Universal Robots URScript: 2024DragonThickMarker.script

def unnamed():
  set_target_payload(1.070000, [0.002000, 0.003000, 0.057000], [0.001723, 0.001723, 0.001723, 0.000000, 0.000000, 0.000000])
  set_tool_communication(True, 1000000, 2, 1, 1.5, 3.5)
  set_tool_output_mode(0)
  set_tool_digital_output_mode(0, 1)
  set_tool_digital_output_mode(1, 1)
  set_tool_voltage(0)
  set_standard_analog_input_domain(0, 1)
  set_standard_analog_input_domain(1, 1)
  set_tool_analog_input_domain(0, 1)
  set_tool_analog_input_domain(1, 1)
  set_analog_outputdomain(0, 0)
  set_analog_outputdomain(1, 0)
  set_input_actions_to_default()
  step_count_120ef5ed_3093_42e9_8e41_c6a461b1e92a = 0.0
  thread Step_Counter_Thread_6ab2a575_f1a7_416e_8c30_f36541ff69b0():
    while (True):
      step_count_120ef5ed_3093_42e9_8e41_c6a461b1e92a = step_count_120ef5ed_3093_42e9_8e41_c6a461b1e92a + 1.0
      sync()
    end
  end
  run Step_Counter_Thread_6ab2a575_f1a7_416e_8c30_f36541ff69b0()
  set_tcp(p[0.0,0.0,0.0,0.0,0.0,0.0])
  set_gravity([0.0, 0.0, 9.82])
  set_safety_mode_transition_hardness(1)
  global Plane_1=p[-0.700006141123905,1.3454883874109249E-6,0.3910559577028425,-1.2089868272251132,-1.2089999932245832,1.20858562628424]
  global Plane_2=p[0.0,0.0,0.0,0.0,0.0,0.0]
  global Point_1=p[0.6913645118948067,-0.12399382748223003,0.49223711947071,-1.2983729986843258,1.1259514972191385,-1.2203503861141718]
  $ 1 "Robot Program"
  $ 2 "Script: 2024Dagonv3_1_marker.script"
  def Machining1():
    # Default parameters:
    global speed_ms = 0.3
    global speed_rads = 0.75
    global accel_mss = 3
    global accel_radss = 1.2
    global blend_radius_m = 0.001

    # Add subprograms here
    # Start of main program
    # Program generated by RoboDK v5.6.5 for UR10e on 12/01/2024 12:52:10
    # Using nominal kinematics.
    blend_radius_m = 0.000
    speed_ms = 1.000
    # set_reference(p[0.335000, -0.152000, -0.035000, 0.000000, 0.000000, 0.000000])
    set_tcp(p[0.000000, 0.000000, 0.252000, 0.000000, 0.000000, 0.000000])
    # Show Tool
    movej([0.067194, -1.029625, -2.540120, -1.142644, 1.570796, 1.637990],accel_radss,speed_rads,0,blend_radius_m)
    movel([0.067194, -1.029625, -2.540120, -1.142644, 1.570796, 1.637990],accel_mss,speed_ms,0,blend_radius_m)
    # Splitting Linear movement in 22 (instruction 7: MoveL 3)
    movel([0.067194, -1.035168, -2.546706, -1.130514, 1.570796, 1.637990],accel_mss,speed_ms,0,blend_radius_m)
    movel([0.067194, -1.040913, -2.553250, -1.118226, 1.570796, 1.637990],accel_mss,speed_ms,0,blend_radius_m)
    movel([0.067194, -1.046863, -2.559752, -1.105774, 1.570796, 1.637990],accel_mss,speed_ms,0,blend_radius_m)
    movel([0.067194, -1.053024, -2.566210, -1.093155, 1.570796, 1.637990],accel_mss,speed_ms,0,blend_radius_m)
    movel([0.067194, -1.059401, -2.572624, -1.080365, 1.570796, 1.637990],accel_mss,speed_ms,0,blend_radius_m)
    movel([0.067194, -1.065999, -2.578992, -1.067399, 1.570796, 1.637990],accel_mss,speed_ms,0,blend_radius_m)
    movel([0.067194, -1.072824, -2.585312, -1.054253, 1.570796, 1.637990],accel_mss,speed_ms,0,blend_radius_m)
    movel([0.067194, -1.079881, -2.591585, -1.040923, 1.570796, 1.637990],accel_mss,speed_ms,0,blend_radius_m)
    movel([0.067194, -1.087175, -2.597809, -1.027405, 1.570796, 1.637990],accel_mss,speed_ms,0,blend_radius_m)
    movel([0.067194, -1.094713, -2.603982, -1.013694, 1.570796, 1.637990],accel_mss,speed_ms,0,blend_radius_m)
    movel([0.067194, -1.102499, -2.610103, -0.999786, 1.570796, 1.637990],accel_mss,speed_ms,0,blend_radius_m)
    movel([0.067194, -1.110540, -2.616171, -0.985677, 1.570796, 1.637990],accel_mss,speed_ms,0,blend_radius_m)
    movel([0.067194, -1.118842, -2.622185, -0.971363, 1.570796, 1.637990],accel_mss,speed_ms,0,blend_radius_m)
    movel([0.067194, -1.127410, -2.628141, -0.956838, 1.570796, 1.637990],accel_mss,speed_ms,0,blend_radius_m)
    movel([0.067194, -1.136249, -2.634040, -0.942099, 1.570796, 1.637990],accel_mss,speed_ms,0,blend_radius_m)
    movel([0.067194, -1.145367, -2.639880, -0.927142, 1.570796, 1.637990],accel_mss,speed_ms,0,blend_radius_m)
    movel([0.067194, -1.154769, -2.645658, -0.911961, 1.570796, 1.637990],accel_mss,speed_ms,0,blend_radius_m)
    movel([0.067194, -1.164461, -2.651374, -0.896554, 1.570796, 1.637990],accel_mss,speed_ms,0,blend_radius_m)
    movel([0.067194, -1.174449, -2.657024, -0.880916, 1.570796, 1.637990],accel_mss,speed_ms,0,blend_radius_m)
    movel([0.067194, -1.184738, -2.662608, -0.865043, 1.570796, 1.637990],accel_mss,speed_ms,0,blend_radius_m)
    movel([0.067194, -1.195335, -2.668122, -0.848931, 1.570796, 1.637990],accel_mss,speed_ms,0,blend_radius_m)
    movel([0.067194, -1.206246, -2.673566, -0.832577, 1.570796, 1.637990],accel_mss,speed_ms,0,blend_radius_m)
    movel([0.067194, -1.206246, -2.673566, -0.832577, 1.570796, 1.637990],accel_mss,speed_ms,0,blend_radius_m)
    speed_ms = 1.000
    movel([0.067194, -1.206246, -2.673566, -0.832577, 1.570796, 1.637990],accel_mss,speed_ms,0,blend_radius_m)
    movel([0.067194, -1.206246, -2.673566, -0.832577, 1.570796, 1.637990],accel_mss,speed_ms,0,blend_radius_m)
    movel([0.067194, -1.206246, -2.673566, -0.832577, 1.570796, 1.637990],accel_mss,speed_ms,0,blend_radius_m)
    speed_ms = 0.005
    # Splitting Linear movement in 4 (instruction 14: MoveL 8)
    movel([0.067194, -1.194262, -2.667574, -0.850553, 1.570796, 1.637990],accel_mss,speed_ms,0,blend_radius_m)
    movel([0.067194, -1.182656, -2.661496, -0.868237, 1.570796, 1.637990],accel_mss,speed_ms,0,blend_radius_m)
    movel([0.067194, -1.171421, -2.655336, -0.885632, 1.570796, 1.637990],accel_mss,speed_ms,0,blend_radius_m)
    movel([0.067194, -1.160549, -2.649095, -0.902745, 1.570796, 1.637990],accel_mss,speed_ms,0,blend_radius_m)
    speed_ms = 1.000
    # Splitting Linear movement in 4 (instruction 16: MoveL 9)
    movel([0.067194, -1.171421, -2.655336, -0.885632, 1.570796, 1.637990],accel_mss,speed_ms,0,blend_radius_m)
    movel([0.067194, -1.182656, -2.661496, -0.868237, 1.570796, 1.637990],accel_mss,speed_ms,0,blend_radius_m)
    movel([0.067194, -1.194262, -2.667574, -0.850553, 1.570796, 1.637990],accel_mss,speed_ms,0,blend_radius_m)
    movel([0.067194, -1.206246, -2.673566, -0.832577, 1.570796, 1.637990],accel_mss,speed_ms,0,blend_radius_m)
    speed_ms = 0.040
    movel([0.067194, -1.206246, -2.673566, -0.832577, 1.570796, 1.637990],accel_mss,speed_ms,0,blend_radius_m)
    speed_ms = 1.000
    movel([0.067194, -1.206246, -2.673566, -0.832577, 1.570796, 1.637990],accel_mss,speed_ms,0,blend_radius_m)
    # Splitting Linear movement in 12 (instruction 21: MoveL 12)
    movel([0.077689, -1.208311, -2.672566, -0.831512, 1.570796, 1.648485],accel_mss,speed_ms,0,blend_radius_m)
    movel([0.088074, -1.210516, -2.671493, -0.830380, 1.570796, 1.658871],accel_mss,speed_ms,0,blend_radius_m)
    movel([0.098348, -1.212858, -2.670347, -0.829184, 1.570796, 1.669145],accel_mss,speed_ms,0,blend_radius_m)
    movel([0.108510, -1.215333, -2.669129, -0.827926, 1.570796, 1.679306],accel_mss,speed_ms,0,blend_radius_m)
    movel([0.118557, -1.217940, -2.667840, -0.826610, 1.570796, 1.689354],accel_mss,speed_ms,0,blend_radius_m)
    movel([0.128491, -1.220675, -2.666478, -0.825236, 1.570796, 1.699287],accel_mss,speed_ms,0,blend_radius_m)
    movel([0.138308, -1.223537, -2.665044, -0.823808, 1.570796, 1.709104],accel_mss,speed_ms,0,blend_radius_m)
    movel([0.148009, -1.226521, -2.663539, -0.822329, 1.570796, 1.718806],accel_mss,speed_ms,0,blend_radius_m)
    movel([0.157594, -1.229625, -2.661962, -0.820802, 1.570796, 1.728390],accel_mss,speed_ms,0,blend_radius_m)
    movel([0.167061, -1.232845, -2.660315, -0.819229, 1.570796, 1.737857],accel_mss,speed_ms,0,blend_radius_m)
    movel([0.176410, -1.236179, -2.658597, -0.817613, 1.570796, 1.747207],accel_mss,speed_ms,0,blend_radius_m)
    movel([0.185641, -1.239624, -2.656808, -0.815957, 1.570796, 1.756438],accel_mss,speed_ms,0,blend_radius_m)
    speed_ms = 0.005
    # Splitting Linear movement in 4 (instruction 23: MoveL 13)
    movel([0.185641, -1.251804, -2.662521, -0.798064, 1.570796, 1.756438],accel_mss,speed_ms,0,blend_radius_m)
    movel([0.185641, -1.264347, -2.668140, -0.779901, 1.570796, 1.756438],accel_mss,speed_ms,0,blend_radius_m)
    movel([0.185641, -1.277260, -2.673664, -0.761465, 1.570796, 1.756438],accel_mss,speed_ms,0,blend_radius_m)
    movel([0.185641, -1.290546, -2.679089, -0.742755, 1.570796, 1.756438],accel_mss,speed_ms,0,blend_radius_m)
    speed_ms = 0.035
    movel([0.190535, -1.290094, -2.679342, -0.742953, 1.570796, 1.761331],accel_mss,speed_ms,0,blend_radius_m)
    movel([0.192211, -1.292754, -2.677845, -0.741789, 1.570796, 1.763007],accel_mss,speed_ms,0,blend_radius_m)
    movel([0.190799, -1.296821, -2.675539, -0.740029, 1.570796, 1.761596],accel_mss,speed_ms,0,blend_radius_m)
    movel([0.186440, -1.300624, -2.673363, -0.738402, 1.570796, 1.757236],accel_mss,speed_ms,0,blend_radius_m)
    speed_ms = 0.005
    movel([0.186440, -1.290042, -2.669080, -0.753268, 1.570796, 1.757236],accel_mss,speed_ms,0,blend_radius_m)
    speed_ms = 0.040
    # Splitting Linear movement in 2 (instruction 32: MoveL 19)
    movel([0.192451, -1.282070, -2.673547, -0.756771, 1.570796, 1.763248],accel_mss,speed_ms,0,blend_radius_m)
    movel([0.198560, -1.273987, -2.677995, -0.760408, 1.570796, 1.769357],accel_mss,speed_ms,0,blend_radius_m)
    speed_ms = 0.005
    movel([0.198560, -1.284689, -2.682355, -0.745345, 1.570796, 1.769357],accel_mss,speed_ms,0,blend_radius_m)
    speed_ms = 0.035
    movel([0.198826, -1.280371, -2.684734, -0.747284, 1.570796, 1.769623],accel_mss,speed_ms,0,blend_radius_m)
    movel([0.195615, -1.278404, -2.685810, -0.748175, 1.570796, 1.766412],accel_mss,speed_ms,0,blend_radius_m)
    movel([0.188967, -1.279617, -2.685147, -0.747625, 1.570796, 1.759764],accel_mss,speed_ms,0,blend_radius_m)
    movel([0.185695, -1.277747, -2.686168, -0.748474, 1.570796, 1.756491],accel_mss,speed_ms,0,blend_radius_m)
    movel([0.186358, -1.274154, -2.688117, -0.750117, 1.570796, 1.757155],accel_mss,speed_ms,0,blend_radius_m)
    movel([0.189422, -1.271170, -2.689724, -0.751495, 1.570796, 1.760218],accel_mss,speed_ms,0,blend_radius_m)
    movel([0.193300, -1.271190, -2.689713, -0.751486, 1.570796, 1.764097],accel_mss,speed_ms,0,blend_radius_m)
    speed_ms = 0.005
    movel([0.193300, -1.260391, -2.685288, -0.766710, 1.570796, 1.764097],accel_mss,speed_ms,0,blend_radius_m)
    speed_ms = 0.040
    # Splitting Linear movement in 4 (instruction 46: MoveL 29)
    movel([0.178839, -1.264011, -2.683369, -0.765009, 1.570796, 1.749636],accel_mss,speed_ms,0,blend_radius_m)
    movel([0.164394, -1.267779, -2.681354, -0.763257, 1.570796, 1.735191],accel_mss,speed_ms,0,blend_radius_m)
    movel([0.149972, -1.271689, -2.679243, -0.761456, 1.570796, 1.720768],accel_mss,speed_ms,0,blend_radius_m)
    movel([0.135577, -1.275738, -2.677038, -0.759613, 1.570796, 1.706373],accel_mss,speed_ms,0,blend_radius_m)
    speed_ms = 0.005
    movel([0.135577, -1.286427, -2.681390, -0.744572, 1.570796, 1.706373],accel_mss,speed_ms,0,blend_radius_m)
    speed_ms = 0.035
    # Splitting Linear movement in 4 (instruction 50: MoveL 31)
    movel([0.144537, -1.281430, -2.684152, -0.746806, 1.570796, 1.715333],accel_mss,speed_ms,0,blend_radius_m)
    movel([0.153562, -1.276433, -2.686883, -0.749073, 1.570796, 1.724358],accel_mss,speed_ms,0,blend_radius_m)
    movel([0.162651, -1.271435, -2.689582, -0.751372, 1.570796, 1.733448],accel_mss,speed_ms,0,blend_radius_m)
    movel([0.171806, -1.266439, -2.692248, -0.753702, 1.570796, 1.742602],accel_mss,speed_ms,0,blend_radius_m)
    # Splitting Linear movement in 2 (instruction 51: MoveL 32)
    movel([0.180931, -1.259543, -2.695876, -0.756970, 1.570796, 1.751728],accel_mss,speed_ms,0,blend_radius_m)
    movel([0.190162, -1.252594, -2.699472, -0.760323, 1.570796, 1.760958],accel_mss,speed_ms,0,blend_radius_m)
    speed_ms = 0.005
    movel([0.190162, -1.241669, -2.694957, -0.775763, 1.570796, 1.760958],accel_mss,speed_ms,0,blend_radius_m)
    speed_ms = 0.040
    # Splitting Linear movement in 8 (instruction 55: MoveL 34)
    movel([0.177847, -1.248567, -2.691444, -0.772378, 1.570796, 1.748643],accel_mss,speed_ms,0,blend_radius_m)
    movel([0.165650, -1.255464, -2.687874, -0.769051, 1.570796, 1.736446],accel_mss,speed_ms,0,blend_radius_m)
    movel([0.153572, -1.262358, -2.684247, -0.765784, 1.570796, 1.724369],accel_mss,speed_ms,0,blend_radius_m)
    movel([0.141614, -1.269247, -2.680564, -0.762579, 1.570796, 1.712411],accel_mss,speed_ms,0,blend_radius_m)
    movel([0.129776, -1.276127, -2.676825, -0.759437, 1.570796, 1.700573],accel_mss,speed_ms,0,blend_radius_m)
    movel([0.118059, -1.282997, -2.673032, -0.756360, 1.570796, 1.688856],accel_mss,speed_ms,0,blend_radius_m)
    movel([0.106463, -1.289855, -2.669185, -0.753349, 1.570796, 1.677259],accel_mss,speed_ms,0,blend_radius_m)
    movel([0.094987, -1.296699, -2.665285, -0.750405, 1.570796, 1.665784],accel_mss,speed_ms,0,blend_radius_m)
    speed_ms = 0.005
    movel([0.094987, -1.307230, -2.669536, -0.735623, 1.570796, 1.665784],accel_mss,speed_ms,0,blend_radius_m)
    speed_ms = 0.035
    movel([0.101831, -1.302246, -2.672429, -0.737715, 1.570796, 1.672627],accel_mss,speed_ms,0,blend_radius_m)
    movel([0.103479, -1.304486, -2.671133, -0.736771, 1.570796, 1.674276],accel_mss,speed_ms,0,blend_radius_m)
    movel([0.102130, -1.311236, -2.667187, -0.733966, 1.570796, 1.672926],accel_mss,speed_ms,0,blend_radius_m)
    # Splitting Linear movement in 2 (instruction 62: MoveL 39)
    movel([0.109636, -1.305912, -2.670304, -0.736173, 1.570796, 1.680433],accel_mss,speed_ms,0,blend_radius_m)
    movel([0.117212, -1.300561, -2.673399, -0.738429, 1.570796, 1.688008],accel_mss,speed_ms,0,blend_radius_m)
    movel([0.121435, -1.299795, -2.673839, -0.738755, 1.570796, 1.692231],accel_mss,speed_ms,0,blend_radius_m)
    speed_ms = 0.005
    movel([0.121435, -1.289206, -2.669552, -0.753631, 1.570796, 1.692231],accel_mss,speed_ms,0,blend_radius_m)
    speed_ms = 0.040
    movel([0.111114, -1.287406, -2.670566, -0.754417, 1.570796, 1.681910],accel_mss,speed_ms,0,blend_radius_m)
    speed_ms = 0.005
    movel([0.111114, -1.298008, -2.674862, -0.739519, 1.570796, 1.681910],accel_mss,speed_ms,0,blend_radius_m)
    speed_ms = 0.035
    movel([0.111474, -1.294449, -2.676887, -0.741053, 1.570796, 1.682270],accel_mss,speed_ms,0,blend_radius_m)
    movel([0.115727, -1.290498, -2.679115, -0.742775, 1.570796, 1.686523],accel_mss,speed_ms,0,blend_radius_m)
    movel([0.120859, -1.291264, -2.678685, -0.742440, 1.570796, 1.691655],accel_mss,speed_ms,0,blend_radius_m)
    movel([0.128037, -1.286245, -2.681491, -0.744653, 1.570796, 1.698833],accel_mss,speed_ms,0,blend_radius_m)
    movel([0.131740, -1.286590, -2.681299, -0.744499, 1.570796, 1.702536],accel_mss,speed_ms,0,blend_radius_m)
    movel([0.132254, -1.290834, -2.678927, -0.742628, 1.570796, 1.703050],accel_mss,speed_ms,0,blend_radius_m)
    speed_ms = 0.005
    movel([0.132254, -1.280177, -2.674597, -0.757615, 1.570796, 1.703050],accel_mss,speed_ms,0,blend_radius_m)
    speed_ms = 0.040
    # Splitting Linear movement in 4 (instruction 80: MoveL 51)
    movel([0.141108, -1.272527, -2.678789, -0.761073, 1.570796, 1.711905],accel_mss,speed_ms,0,blend_radius_m)
    movel([0.150084, -1.264799, -2.682949, -0.764641, 1.570796, 1.720881],accel_mss,speed_ms,0,blend_radius_m)
    movel([0.159184, -1.256990, -2.687076, -0.768323, 1.570796, 1.729980],accel_mss,speed_ms,0,blend_radius_m)
    movel([0.168409, -1.249099, -2.691171, -0.772119, 1.570796, 1.739205],accel_mss,speed_ms,0,blend_radius_m)
    speed_ms = 0.005
    movel([0.168409, -1.259975, -2.695651, -0.756764, 1.570796, 1.739205],accel_mss,speed_ms,0,blend_radius_m)
    speed_ms = 0.035
    movel([0.155366, -1.269180, -2.690789, -0.752420, 1.570796, 1.726162],accel_mss,speed_ms,0,blend_radius_m)
    movel([0.143271, -1.278387, -2.685819, -0.748183, 1.570796, 1.714067],accel_mss,speed_ms,0,blend_radius_m)
    speed_ms = 0.005
    movel([0.143271, -1.267639, -2.681429, -0.763321, 1.570796, 1.714067],accel_mss,speed_ms,0,blend_radius_m)
    speed_ms = 0.040
    # Splitting Linear movement in 4 (instruction 89: MoveL 56)
    movel([0.142087, -1.279264, -2.675101, -0.758024, 1.570796, 1.712884],accel_mss,speed_ms,0,blend_radius_m)
    movel([0.140935, -1.290667, -2.668725, -0.752996, 1.570796, 1.711731],accel_mss,speed_ms,0,blend_radius_m)
    movel([0.139813, -1.301859, -2.662303, -0.748227, 1.570796, 1.710609],accel_mss,speed_ms,0,blend_radius_m)
    movel([0.138719, -1.312847, -2.655836, -0.743706, 1.570796, 1.709516],accel_mss,speed_ms,0,blend_radius_m)
    speed_ms = 0.005
    movel([0.138719, -1.323250, -2.660010, -0.729129, 1.570796, 1.709516],accel_mss,speed_ms,0,blend_radius_m)
    speed_ms = 0.035
    movel([0.151265, -1.322547, -2.660435, -0.729407, 1.570796, 1.722061],accel_mss,speed_ms,0,blend_radius_m)
    movel([0.161811, -1.317841, -2.663266, -0.731282, 1.570796, 1.732607],accel_mss,speed_ms,0,blend_radius_m)
    movel([0.171157, -1.310457, -2.667645, -0.734287, 1.570796, 1.741953],accel_mss,speed_ms,0,blend_radius_m)
    movel([0.178358, -1.301250, -2.673002, -0.738136, 1.570796, 1.749154],accel_mss,speed_ms,0,blend_radius_m)
    movel([0.182387, -1.291138, -2.678756, -0.742495, 1.570796, 1.753183],accel_mss,speed_ms,0,blend_radius_m)
    movel([0.182560, -1.283536, -2.682993, -0.745861, 1.570796, 1.753356],accel_mss,speed_ms,0,blend_radius_m)
    # Splitting Linear movement in 2 (instruction 99: MoveL 64)
    movel([0.178714, -1.278759, -2.685616, -0.748014, 1.570796, 1.749511],accel_mss,speed_ms,0,blend_radius_m)
    movel([0.174816, -1.273981, -2.688211, -0.750197, 1.570796, 1.745613],accel_mss,speed_ms,0,blend_radius_m)
    movel([0.167634, -1.272793, -2.688852, -0.750745, 1.570796, 1.738430],accel_mss,speed_ms,0,blend_radius_m)
    speed_ms = 0.005
    movel([0.167634, -1.262005, -2.684434, -0.765950, 1.570796, 1.738430],accel_mss,speed_ms,0,blend_radius_m)
    speed_ms = 0.040
    # Splitting Linear movement in 6 (instruction 104: MoveL 67)
    movel([0.162362, -1.272295, -2.678915, -0.761179, 1.570796, 1.733159],accel_mss,speed_ms,0,blend_radius_m)
    movel([0.157203, -1.282396, -2.673366, -0.756626, 1.570796, 1.727999],accel_mss,speed_ms,0,blend_radius_m)
    movel([0.152152, -1.292315, -2.667790, -0.752284, 1.570796, 1.722948],accel_mss,speed_ms,0,blend_radius_m)
    movel([0.147205, -1.302059, -2.662187, -0.748143, 1.570796, 1.718002],accel_mss,speed_ms,0,blend_radius_m)
    movel([0.142361, -1.311633, -2.656558, -0.744198, 1.570796, 1.713157],accel_mss,speed_ms,0,blend_radius_m)
    movel([0.137614, -1.321044, -2.650904, -0.740440, 1.570796, 1.708410],accel_mss,speed_ms,0,blend_radius_m)
    speed_ms = 0.005
    movel([0.137614, -1.331380, -2.655040, -0.725969, 1.570796, 1.708410],accel_mss,speed_ms,0,blend_radius_m)
    speed_ms = 0.035
    movel([0.130829, -1.332244, -2.654506, -0.725639, 1.570796, 1.701625],accel_mss,speed_ms,0,blend_radius_m)
    movel([0.121495, -1.338806, -2.650419, -0.723164, 1.570796, 1.692292],accel_mss,speed_ms,0,blend_radius_m)
    movel([0.117433, -1.347747, -2.644752, -0.719890, 1.570796, 1.688229],accel_mss,speed_ms,0,blend_radius_m)
    movel([0.120880, -1.353838, -2.640825, -0.717726, 1.570796, 1.691677],accel_mss,speed_ms,0,blend_radius_m)
    movel([0.129722, -1.353699, -2.640916, -0.717775, 1.570796, 1.700518],accel_mss,speed_ms,0,blend_radius_m)
    movel([0.135832, -1.350295, -2.643116, -0.718978, 1.570796, 1.706628],accel_mss,speed_ms,0,blend_radius_m)
    movel([0.140541, -1.345317, -2.646304, -0.720769, 1.570796, 1.711337],accel_mss,speed_ms,0,blend_radius_m)
    speed_ms = 0.005
    movel([0.140541, -1.335099, -2.642235, -0.735055, 1.570796, 1.711337],accel_mss,speed_ms,0,blend_radius_m)
    speed_ms = 0.040
    # Splitting Linear movement in 4 (instruction 118: MoveL 77)
    movel([0.141902, -1.345385, -2.635715, -0.731290, 1.570796, 1.712698],accel_mss,speed_ms,0,blend_radius_m)
    movel([0.143229, -1.355523, -2.629141, -0.727725, 1.570796, 1.714025],accel_mss,speed_ms,0,blend_radius_m)
    movel([0.144523, -1.365518, -2.622515, -0.724355, 1.570796, 1.715319],accel_mss,speed_ms,0,blend_radius_m)
    movel([0.145785, -1.375375, -2.615839, -0.721176, 1.570796, 1.716582],accel_mss,speed_ms,0,blend_radius_m)
    speed_ms = 0.005
    movel([0.145785, -1.385238, -2.619719, -0.707432, 1.570796, 1.716582],accel_mss,speed_ms,0,blend_radius_m)
    speed_ms = 0.035
    movel([0.152329, -1.384002, -2.620578, -0.707809, 1.570796, 1.723125],accel_mss,speed_ms,0,blend_radius_m)
    movel([0.160842, -1.377593, -2.624993, -0.709803, 1.570796, 1.731638],accel_mss,speed_ms,0,blend_radius_m)
    movel([0.164107, -1.369156, -2.630712, -0.712521, 1.570796, 1.734903],accel_mss,speed_ms,0,blend_radius_m)
    movel([0.160071, -1.363662, -2.634378, -0.714348, 1.570796, 1.730868],accel_mss,speed_ms,0,blend_radius_m)
    movel([0.151027, -1.364502, -2.633821, -0.714066, 1.570796, 1.721824],accel_mss,speed_ms,0,blend_radius_m)
    movel([0.145179, -1.368216, -2.631342, -0.712831, 1.570796, 1.715975],accel_mss,speed_ms,0,blend_radius_m)
    movel([0.141048, -1.373192, -2.627989, -0.711208, 1.570796, 1.711845],accel_mss,speed_ms,0,blend_radius_m)
    speed_ms = 0.005
    movel([0.141048, -1.363219, -2.624052, -0.725117, 1.570796, 1.711845],accel_mss,speed_ms,0,blend_radius_m)
    speed_ms = 0.040
    # Splitting Linear movement in 4 (instruction 132: MoveL 87)
    movel([0.138960, -1.371507, -2.618475, -0.722406, 1.570796, 1.709756],accel_mss,speed_ms,0,blend_radius_m)
    movel([0.136912, -1.379679, -2.612878, -0.719832, 1.570796, 1.707708],accel_mss,speed_ms,0,blend_radius_m)
    movel([0.134903, -1.387739, -2.607259, -0.717391, 1.570796, 1.705699],accel_mss,speed_ms,0,blend_radius_m)
    movel([0.132931, -1.395690, -2.601621, -0.715078, 1.570796, 1.703727],accel_mss,speed_ms,0,blend_radius_m)
    speed_ms = 0.005
    movel([0.132931, -1.405366, -2.605409, -0.701614, 1.570796, 1.703727],accel_mss,speed_ms,0,blend_radius_m)
    speed_ms = 0.035
    movel([0.133810, -1.412569, -2.600136, -0.699684, 1.570796, 1.704607],accel_mss,speed_ms,0,blend_radius_m)
    movel([0.131777, -1.420121, -2.594521, -0.697747, 1.570796, 1.702574],accel_mss,speed_ms,0,blend_radius_m)
    movel([0.127141, -1.427318, -2.589086, -0.695985, 1.570796, 1.697937],accel_mss,speed_ms,0,blend_radius_m)
    movel([0.120176, -1.433518, -2.584338, -0.694533, 1.570796, 1.690972],accel_mss,speed_ms,0,blend_radius_m)
    # Splitting Linear movement in 2 (instruction 140: MoveL 93)
    movel([0.112265, -1.436686, -2.581888, -0.693815, 1.570796, 1.683061],accel_mss,speed_ms,0,blend_radius_m)
    movel([0.104390, -1.439876, -2.579405, -0.693108, 1.570796, 1.675186],accel_mss,speed_ms,0,blend_radius_m)
    speed_ms = 0.005
    movel([0.104390, -1.430531, -2.575774, -0.706084, 1.570796, 1.675186],accel_mss,speed_ms,0,blend_radius_m)
    speed_ms = 0.040
    movel([0.093930, -1.437280, -2.570548, -0.704561, 1.570796, 1.664726],accel_mss,speed_ms,0,blend_radius_m)
    speed_ms = 0.005
    movel([0.093930, -1.446561, -2.574149, -0.691679, 1.570796, 1.664726],accel_mss,speed_ms,0,blend_radius_m)
    speed_ms = 0.035
    movel([0.090838, -1.453615, -2.568524, -0.690250, 1.570796, 1.661634],accel_mss,speed_ms,0,blend_radius_m)
    movel([0.093532, -1.458384, -2.564675, -0.689330, 1.570796, 1.664329],accel_mss,speed_ms,0,blend_radius_m)
    movel([0.100282, -1.458870, -2.564281, -0.689238, 1.570796, 1.671079],accel_mss,speed_ms,0,blend_radius_m)
    movel([0.109545, -1.452972, -2.569040, -0.690377, 1.570796, 1.680341],accel_mss,speed_ms,0,blend_radius_m)
    speed_ms = 0.005
    movel([0.109545, -1.443754, -2.565467, -0.703168, 1.570796, 1.680341],accel_mss,speed_ms,0,blend_radius_m)
    speed_ms = 0.040
    # Splitting Linear movement in 4 (instruction 155: MoveL 102)
    movel([0.105118, -1.454139, -2.557178, -0.701072, 1.570796, 1.675915],accel_mss,speed_ms,0,blend_radius_m)
    movel([0.100797, -1.464350, -2.548859, -0.699180, 1.570796, 1.671593],accel_mss,speed_ms,0,blend_radius_m)
    movel([0.096577, -1.474395, -2.540509, -0.697484, 1.570796, 1.667373],accel_mss,speed_ms,0,blend_radius_m)
    movel([0.092455, -1.484282, -2.532131, -0.695975, 1.570796, 1.663251],accel_mss,speed_ms,0,blend_radius_m)
    speed_ms = 0.005
    movel([0.092455, -1.493102, -2.535530, -0.683756, 1.570796, 1.663251],accel_mss,speed_ms,0,blend_radius_m)
    speed_ms = 0.035
    # Splitting Linear movement in 4 (instruction 159: MoveL 104)
    movel([0.096922, -1.486423, -2.541293, -0.684673, 1.570796, 1.667719],accel_mss,speed_ms,0,blend_radius_m)
    movel([0.101459, -1.479672, -2.547041, -0.685676, 1.570796, 1.672255],accel_mss,speed_ms,0,blend_radius_m)
    movel([0.106066, -1.472850, -2.552774, -0.686766, 1.570796, 1.676862],accel_mss,speed_ms,0,blend_radius_m)
    movel([0.110745, -1.465952, -2.558491, -0.687945, 1.570796, 1.681541],accel_mss,speed_ms,0,blend_radius_m)
    speed_ms = 0.005
    movel([0.110745, -1.456863, -2.554975, -0.700551, 1.570796, 1.681541],accel_mss,speed_ms,0,blend_radius_m)
    speed_ms = 0.040
    # Splitting Linear movement in 4 (instruction 163: MoveL 106)
    movel([0.117751, -1.462174, -2.550646, -0.699569, 1.570796, 1.688548],accel_mss,speed_ms,0,blend_radius_m)
    movel([0.124645, -1.467519, -2.546242, -0.698628, 1.570796, 1.695441],accel_mss,speed_ms,0,blend_radius_m)
    movel([0.131427, -1.472898, -2.541765, -0.697727, 1.570796, 1.702223],accel_mss,speed_ms,0,blend_radius_m)
    movel([0.138099, -1.478306, -2.537215, -0.696868, 1.570796, 1.708895],accel_mss,speed_ms,0,blend_radius_m)
    speed_ms = 0.005
    movel([0.138099, -1.487185, -2.540639, -0.684565, 1.570796, 1.708895],accel_mss,speed_ms,0,blend_radius_m)
    speed_ms = 0.035
    # Splitting Linear movement in 4 (instruction 167: MoveL 108)
    movel([0.127868, -1.489358, -2.538770, -0.684261, 1.570796, 1.698664],accel_mss,speed_ms,0,blend_radius_m)
    movel([0.117652, -1.491602, -2.536831, -0.683956, 1.570796, 1.688448],accel_mss,speed_ms,0,blend_radius_m)
    movel([0.107454, -1.493915, -2.534825, -0.683650, 1.570796, 1.678250],accel_mss,speed_ms,0,blend_radius_m)
    movel([0.097275, -1.496295, -2.532750, -0.683344, 1.570796, 1.668071],accel_mss,speed_ms,0,blend_radius_m)
    speed_ms = 0.005
    movel([0.097275, -1.487507, -2.529364, -0.695518, 1.570796, 1.668071],accel_mss,speed_ms,0,blend_radius_m)
    speed_ms = 0.040
    # Splitting Linear movement in 4 (instruction 171: MoveL 110)
    movel([0.107634, -1.482776, -2.533418, -0.696195, 1.570796, 1.678430],accel_mss,speed_ms,0,blend_radius_m)
    movel([0.118073, -1.478075, -2.537410, -0.696904, 1.570796, 1.688869],accel_mss,speed_ms,0,blend_radius_m)
    movel([0.128591, -1.473404, -2.541341, -0.697644, 1.570796, 1.699387],accel_mss,speed_ms,0,blend_radius_m)
    movel([0.139188, -1.468765, -2.545209, -0.698415, 1.570796, 1.709984],accel_mss,speed_ms,0,blend_radius_m)
    speed_ms = 0.005
    movel([0.139188, -1.477738, -2.548674, -0.685977, 1.570796, 1.709984],accel_mss,speed_ms,0,blend_radius_m)
    speed_ms = 0.035
    # Splitting Linear movement in 4 (instruction 175: MoveL 112)
    movel([0.132091, -1.479248, -2.547400, -0.685741, 1.570796, 1.702887],accel_mss,speed_ms,0,blend_radius_m)
    movel([0.125000, -1.480792, -2.546093, -0.685504, 1.570796, 1.695797],accel_mss,speed_ms,0,blend_radius_m)
    movel([0.117917, -1.482369, -2.544754, -0.685266, 1.570796, 1.688714],accel_mss,speed_ms,0,blend_radius_m)
    movel([0.110843, -1.483979, -2.543382, -0.685027, 1.570796, 1.681639],accel_mss,speed_ms,0,blend_radius_m)
    # Splitting Linear movement in 4 (instruction 176: MoveL 113)
    movel([0.114286, -1.478824, -2.547758, -0.685807, 1.570796, 1.685082],accel_mss,speed_ms,0,blend_radius_m)
    movel([0.117770, -1.473627, -2.552124, -0.686637, 1.570796, 1.688566],accel_mss,speed_ms,0,blend_radius_m)
    movel([0.121295, -1.468387, -2.556482, -0.687520, 1.570796, 1.692091],accel_mss,speed_ms,0,blend_radius_m)
    movel([0.124862, -1.463102, -2.560831, -0.688456, 1.570796, 1.695658],accel_mss,speed_ms,0,blend_radius_m)
    movel([0.127311, -1.460587, -2.562885, -0.688917, 1.570796, 1.698107],accel_mss,speed_ms,0,blend_radius_m)
    movel([0.133759, -1.460021, -2.563346, -0.689022, 1.570796, 1.704556],accel_mss,speed_ms,0,blend_radius_m)
    movel([0.134542, -1.462829, -2.561055, -0.688505, 1.570796, 1.705338],accel_mss,speed_ms,0,blend_radius_m)
    # Splitting Linear movement in 2 (instruction 180: MoveL 117)
    movel([0.133599, -1.469513, -2.555549, -0.687326, 1.570796, 1.704396],accel_mss,speed_ms,0,blend_radius_m)
    movel([0.132673, -1.476129, -2.550028, -0.686232, 1.570796, 1.703469],accel_mss,speed_ms,0,blend_radius_m)
    speed_ms = 0.005
    movel([0.132673, -1.467140, -2.546556, -0.698693, 1.570796, 1.703469],accel_mss,speed_ms,0,blend_radius_m)
    speed_ms = 0.040
    # Splitting Linear movement in 2 (instruction 184: MoveL 119)
    movel([0.131362, -1.475209, -2.539826, -0.697354, 1.570796, 1.702158],accel_mss,speed_ms,0,blend_radius_m)
    movel([0.130076, -1.483180, -2.533073, -0.696136, 1.570796, 1.700873],accel_mss,speed_ms,0,blend_radius_m)
    speed_ms = 0.005
    movel([0.130076, -1.492011, -2.536477, -0.683901, 1.570796, 1.700873],accel_mss,speed_ms,0,blend_radius_m)
    speed_ms = 0.035
    # Splitting Linear movement in 2 (instruction 188: MoveL 121)
    movel([0.129165, -1.497777, -2.531454, -0.683159, 1.570796, 1.699962],accel_mss,speed_ms,0,blend_radius_m)
    movel([0.128267, -1.503492, -2.526419, -0.682478, 1.570796, 1.699064],accel_mss,speed_ms,0,blend_radius_m)
    speed_ms = 0.005
    movel([0.128267, -1.494776, -2.523063, -0.694550, 1.570796, 1.699064],accel_mss,speed_ms,0,blend_radius_m)
    speed_ms = 0.040
    # Splitting Linear movement in 4 (instruction 192: MoveL 123)
    movel([0.126085, -1.501282, -2.517350, -0.693757, 1.570796, 1.696881],accel_mss,speed_ms,0,blend_radius_m)
    movel([0.123936, -1.507725, -2.511623, -0.693041, 1.570796, 1.694732],accel_mss,speed_ms,0,blend_radius_m)
    movel([0.121820, -1.514105, -2.505884, -0.692400, 1.570796, 1.692616],accel_mss,speed_ms,0,blend_radius_m)
    movel([0.119736, -1.520424, -2.500133, -0.691832, 1.570796, 1.690532],accel_mss,speed_ms,0,blend_radius_m)
    speed_ms = 0.005
    movel([0.119736, -1.528887, -2.503384, -0.680118, 1.570796, 1.690532],accel_mss,speed_ms,0,blend_radius_m)
    speed_ms = 0.035
    movel([0.126505, -1.525050, -2.506934, -0.680405, 1.570796, 1.697301],accel_mss,speed_ms,0,blend_radius_m)
    movel([0.132226, -1.524886, -2.507085, -0.680417, 1.570796, 1.703022],accel_mss,speed_ms,0,blend_radius_m)
    speed_ms = 0.005
    movel([0.132226, -1.516384, -2.503818, -0.692187, 1.570796, 1.703022],accel_mss,speed_ms,0,blend_radius_m)
    speed_ms = 0.040
    # Splitting Linear movement in 2 (instruction 201: MoveL 128)
    movel([0.122788, -1.516132, -2.504047, -0.692210, 1.570796, 1.693584],accel_mss,speed_ms,0,blend_radius_m)
    movel([0.113311, -1.515963, -2.504200, -0.692226, 1.570796, 1.684107],accel_mss,speed_ms,0,blend_radius_m)
    speed_ms = 0.005
    movel([0.113311, -1.524470, -2.507469, -0.680450, 1.570796, 1.684107],accel_mss,speed_ms,0,blend_radius_m)
    speed_ms = 0.035
    movel([0.119444, -1.519667, -2.511873, -0.680849, 1.570796, 1.690241],accel_mss,speed_ms,0,blend_radius_m)
    movel([0.127561, -1.516834, -2.514453, -0.681102, 1.570796, 1.698358],accel_mss,speed_ms,0,blend_radius_m)
    movel([0.133553, -1.516376, -2.514869, -0.681144, 1.570796, 1.704350],accel_mss,speed_ms,0,blend_radius_m)
    movel([0.139808, -1.514237, -2.516806, -0.681346, 1.570796, 1.710604],accel_mss,speed_ms,0,blend_radius_m)
    movel([0.143696, -1.509524, -2.521046, -0.681819, 1.570796, 1.714492],accel_mss,speed_ms,0,blend_radius_m)
    movel([0.143666, -1.506404, -2.523833, -0.682152, 1.570796, 1.714462],accel_mss,speed_ms,0,blend_radius_m)
    movel([0.140353, -1.503852, -2.526100, -0.682437, 1.570796, 1.711150],accel_mss,speed_ms,0,blend_radius_m)
    speed_ms = 0.005
    movel([0.140353, -1.495139, -2.522746, -0.694503, 1.570796, 1.711150],accel_mss,speed_ms,0,blend_radius_m)
    speed_ms = 0.040
    # Splitting Linear movement in 10 (instruction 215: MoveL 138)
    movel([0.136503, -1.488144, -2.528815, -0.695430, 1.570796, 1.707299],accel_mss,speed_ms,0,blend_radius_m)
    movel([0.132578, -1.481116, -2.534832, -0.696441, 1.570796, 1.703374],accel_mss,speed_ms,0,blend_radius_m)
    movel([0.128576, -1.474055, -2.540795, -0.697539, 1.570796, 1.699372],accel_mss,speed_ms,0,blend_radius_m)
    movel([0.124495, -1.466962, -2.546703, -0.698724, 1.570796, 1.695292],accel_mss,speed_ms,0,blend_radius_m)
    movel([0.120334, -1.459836, -2.552557, -0.699996, 1.570796, 1.691130],accel_mss,speed_ms,0,blend_radius_m)
    movel([0.116090, -1.452679, -2.558354, -0.701356, 1.570796, 1.686886],accel_mss,speed_ms,0,blend_radius_m)
    movel([0.111760, -1.445489, -2.564094, -0.702805, 1.570796, 1.682557],accel_mss,speed_ms,0,blend_radius_m)
    movel([0.107344, -1.438269, -2.569776, -0.704344, 1.570796, 1.678140],accel_mss,speed_ms,0,blend_radius_m)
    movel([0.102838, -1.431017, -2.575400, -0.705972, 1.570796, 1.673635],accel_mss,speed_ms,0,blend_radius_m)
    movel([0.098241, -1.423736, -2.580963, -0.707690, 1.570796, 1.669037],accel_mss,speed_ms,0,blend_radius_m)
    speed_ms = 0.005
    movel([0.098241, -1.433146, -2.584624, -0.694618, 1.570796, 1.669037],accel_mss,speed_ms,0,blend_radius_m)
    speed_ms = 0.035
    movel([0.087607, -1.439125, -2.579991, -0.693273, 1.570796, 1.658404],accel_mss,speed_ms,0,blend_radius_m)
    movel([0.079985, -1.447477, -2.573423, -0.691489, 1.570796, 1.650781],accel_mss,speed_ms,0,blend_radius_m)
    movel([0.076763, -1.456675, -2.566059, -0.689655, 1.570796, 1.647559],accel_mss,speed_ms,0,blend_radius_m)
    # Splitting Linear movement in 2 (instruction 222: MoveL 143)
    movel([0.077988, -1.461010, -2.562540, -0.688839, 1.570796, 1.648784],accel_mss,speed_ms,0,blend_radius_m)
    movel([0.079198, -1.465323, -2.559009, -0.688057, 1.570796, 1.649994],accel_mss,speed_ms,0,blend_radius_m)
    movel([0.085673, -1.469620, -2.555461, -0.687308, 1.570796, 1.656469],accel_mss,speed_ms,0,blend_radius_m)
    movel([0.091200, -1.470506, -2.554726, -0.687158, 1.570796, 1.661996],accel_mss,speed_ms,0,blend_radius_m)
    movel([0.098089, -1.469488, -2.555571, -0.687331, 1.570796, 1.668885],accel_mss,speed_ms,0,blend_radius_m)
    # Splitting Linear movement in 2 (instruction 226: MoveL 147)
    movel([0.104128, -1.466423, -2.558104, -0.687862, 1.570796, 1.674924],accel_mss,speed_ms,0,blend_radius_m)
    movel([0.110198, -1.463363, -2.560618, -0.688408, 1.570796, 1.680994],accel_mss,speed_ms,0,blend_radius_m)
    movel([0.119150, -1.454254, -2.568010, -0.690125, 1.570796, 1.689947],accel_mss,speed_ms,0,blend_radius_m)
    movel([0.129208, -1.447858, -2.573121, -0.691410, 1.570796, 1.700004],accel_mss,speed_ms,0,blend_radius_m)
    # Splitting Linear movement in 2 (instruction 229: MoveL 150)
    movel([0.135129, -1.447122, -2.573705, -0.691563, 1.570796, 1.705926],accel_mss,speed_ms,0,blend_radius_m)
    movel([0.141047, -1.446414, -2.574265, -0.691710, 1.570796, 1.711843],accel_mss,speed_ms,0,blend_radius_m)
    movel([0.146886, -1.449933, -2.571470, -0.690986, 1.570796, 1.717683],accel_mss,speed_ms,0,blend_radius_m)
    # Splitting Linear movement in 2 (instruction 231: MoveL 152)
    movel([0.147893, -1.454749, -2.567612, -0.690028, 1.570796, 1.718689],accel_mss,speed_ms,0,blend_radius_m)
    movel([0.148887, -1.459536, -2.563740, -0.689113, 1.570796, 1.719683],accel_mss,speed_ms,0,blend_radius_m)
    # Splitting Linear movement in 6 (instruction 232: MoveL 153)
    movel([0.147642, -1.466517, -2.558027, -0.687846, 1.570796, 1.718438],accel_mss,speed_ms,0,blend_radius_m)
    movel([0.146418, -1.473421, -2.552297, -0.686671, 1.570796, 1.717214],accel_mss,speed_ms,0,blend_radius_m)
    movel([0.145215, -1.480251, -2.546551, -0.685587, 1.570796, 1.716011],accel_mss,speed_ms,0,blend_radius_m)
    movel([0.144031, -1.487009, -2.540790, -0.684590, 1.570796, 1.714828],accel_mss,speed_ms,0,blend_radius_m)
    movel([0.142868, -1.493698, -2.535013, -0.683678, 1.570796, 1.713664],accel_mss,speed_ms,0,blend_radius_m)
    movel([0.141723, -1.500319, -2.529221, -0.682849, 1.570796, 1.712520],accel_mss,speed_ms,0,blend_radius_m)
    speed_ms = 0.005
    movel([0.141723, -1.491571, -2.525852, -0.694966, 1.570796, 1.712520],accel_mss,speed_ms,0,blend_radius_m)
    speed_ms = 0.040
    # Splitting Linear movement in 12 (instruction 236: MoveL 155)
    movel([0.138463, -1.484988, -2.531527, -0.695874, 1.570796, 1.709259],accel_mss,speed_ms,0,blend_radius_m)
    movel([0.135143, -1.478372, -2.537159, -0.696858, 1.570796, 1.705939],accel_mss,speed_ms,0,blend_radius_m)
    movel([0.131763, -1.471723, -2.542747, -0.697919, 1.570796, 1.702559],accel_mss,speed_ms,0,blend_radius_m)
    movel([0.128321, -1.465039, -2.548291, -0.699059, 1.570796, 1.699117],accel_mss,speed_ms,0,blend_radius_m)
    movel([0.124815, -1.458321, -2.553791, -0.700277, 1.570796, 1.695611],accel_mss,speed_ms,0,blend_radius_m)
    movel([0.121244, -1.451570, -2.559245, -0.701574, 1.570796, 1.692040],accel_mss,speed_ms,0,blend_radius_m)
    movel([0.117606, -1.444785, -2.564652, -0.702952, 1.570796, 1.688402],accel_mss,speed_ms,0,blend_radius_m)
    movel([0.113900, -1.437966, -2.570013, -0.704410, 1.570796, 1.684696],accel_mss,speed_ms,0,blend_radius_m)
    movel([0.110124, -1.431113, -2.575326, -0.705950, 1.570796, 1.680920],accel_mss,speed_ms,0,blend_radius_m)
    movel([0.106276, -1.424226, -2.580591, -0.707572, 1.570796, 1.677073],accel_mss,speed_ms,0,blend_radius_m)
    movel([0.102355, -1.417306, -2.585806, -0.709277, 1.570796, 1.673151],accel_mss,speed_ms,0,blend_radius_m)
    movel([0.098359, -1.410353, -2.590972, -0.711064, 1.570796, 1.669155],accel_mss,speed_ms,0,blend_radius_m)
    speed_ms = 0.005
    movel([0.098359, -1.419891, -2.594693, -0.697805, 1.570796, 1.669155],accel_mss,speed_ms,0,blend_radius_m)
    speed_ms = 0.035
    movel([0.101696, -1.415163, -2.598217, -0.699008, 1.570796, 1.672492],accel_mss,speed_ms,0,blend_radius_m)
    movel([0.106933, -1.411351, -2.601033, -0.700004, 1.570796, 1.677730],accel_mss,speed_ms,0,blend_radius_m)
    movel([0.115800, -1.409702, -2.602245, -0.700442, 1.570796, 1.686597],accel_mss,speed_ms,0,blend_radius_m)
    movel([0.120673, -1.414057, -2.599037, -0.699295, 1.570796, 1.691469],accel_mss,speed_ms,0,blend_radius_m)
    movel([0.118728, -1.421731, -2.593312, -0.697346, 1.570796, 1.689524],accel_mss,speed_ms,0,blend_radius_m)
    movel([0.111240, -1.428174, -2.588434, -0.695781, 1.570796, 1.682037],accel_mss,speed_ms,0,blend_radius_m)
    movel([0.104920, -1.429900, -2.587116, -0.695373, 1.570796, 1.675716],accel_mss,speed_ms,0,blend_radius_m)
    speed_ms = 0.005
    movel([0.104920, -1.420458, -2.583440, -0.708491, 1.570796, 1.675716],accel_mss,speed_ms,0,blend_radius_m)
    speed_ms = 0.040
    # Splitting Linear movement in 4 (instruction 250: MoveL 165)
    movel([0.099541, -1.417802, -2.585435, -0.709152, 1.570796, 1.670337],accel_mss,speed_ms,0,blend_radius_m)
    movel([0.094114, -1.415175, -2.587397, -0.709817, 1.570796, 1.664910],accel_mss,speed_ms,0,blend_radius_m)
    movel([0.088638, -1.412579, -2.589326, -0.710484, 1.570796, 1.659435],accel_mss,speed_ms,0,blend_radius_m)
    movel([0.083114, -1.410015, -2.591221, -0.711153, 1.570796, 1.653910],accel_mss,speed_ms,0,blend_radius_m)
    speed_ms = 0.005
    movel([0.083114, -1.419556, -2.594944, -0.697889, 1.570796, 1.653910],accel_mss,speed_ms,0,blend_radius_m)
    speed_ms = 0.035
    movel([0.089884, -1.410118, -2.601940, -0.700331, 1.570796, 1.660680],accel_mss,speed_ms,0,blend_radius_m)
    movel([0.096591, -1.403663, -2.606644, -0.702082, 1.570796, 1.667387],accel_mss,speed_ms,0,blend_radius_m)
    movel([0.106973, -1.397613, -2.610995, -0.703781, 1.570796, 1.677770],accel_mss,speed_ms,0,blend_radius_m)
    movel([0.118175, -1.394764, -2.613024, -0.704601, 1.570796, 1.688972],accel_mss,speed_ms,0,blend_radius_m)
    # Splitting Linear movement in 4 (instruction 258: MoveL 171)
    movel([0.123682, -1.395876, -2.612234, -0.704280, 1.570796, 1.694479],accel_mss,speed_ms,0,blend_radius_m)
    movel([0.129160, -1.397020, -2.611418, -0.703951, 1.570796, 1.699957],accel_mss,speed_ms,0,blend_radius_m)
    movel([0.134609, -1.398197, -2.610577, -0.703615, 1.570796, 1.705405],accel_mss,speed_ms,0,blend_radius_m)
    movel([0.140028, -1.399407, -2.609711, -0.703272, 1.570796, 1.710824],accel_mss,speed_ms,0,blend_radius_m)
    movel([0.148049, -1.398606, -2.610285, -0.703499, 1.570796, 1.718846],accel_mss,speed_ms,0,blend_radius_m)
    movel([0.156488, -1.395608, -2.612424, -0.704357, 1.570796, 1.727284],accel_mss,speed_ms,0,blend_radius_m)
    movel([0.164706, -1.390550, -2.616003, -0.705836, 1.570796, 1.735503],accel_mss,speed_ms,0,blend_radius_m)
    # Splitting Linear movement in 2 (instruction 262: MoveL 175)
    movel([0.170815, -1.383589, -2.620864, -0.707936, 1.570796, 1.741611],accel_mss,speed_ms,0,blend_radius_m)
    movel([0.177013, -1.376549, -2.625707, -0.710134, 1.570796, 1.747809],accel_mss,speed_ms,0,blend_radius_m)
    movel([0.180329, -1.368166, -2.631376, -0.712847, 1.570796, 1.751126],accel_mss,speed_ms,0,blend_radius_m)
    movel([0.180574, -1.359663, -2.637020, -0.715706, 1.570796, 1.751370],accel_mss,speed_ms,0,blend_radius_m)
    movel([0.177774, -1.353790, -2.640857, -0.717743, 1.570796, 1.748570],accel_mss,speed_ms,0,blend_radius_m)
    movel([0.172376, -1.350087, -2.643250, -0.719052, 1.570796, 1.743173],accel_mss,speed_ms,0,blend_radius_m)
    movel([0.164952, -1.348798, -2.644078, -0.719513, 1.570796, 1.735748],accel_mss,speed_ms,0,blend_radius_m)
    movel([0.156125, -1.350121, -2.643228, -0.719040, 1.570796, 1.726922],accel_mss,speed_ms,0,blend_radius_m)
    movel([0.146546, -1.354226, -2.640573, -0.717589, 1.570796, 1.717342],accel_mss,speed_ms,0,blend_radius_m)
    movel([0.137861, -1.360452, -2.636500, -0.715436, 1.570796, 1.708658],accel_mss,speed_ms,0,blend_radius_m)
    movel([0.130795, -1.368120, -2.631407, -0.712862, 1.570796, 1.701591],accel_mss,speed_ms,0,blend_radius_m)
    movel([0.126015, -1.376578, -2.625687, -0.710124, 1.570796, 1.696812],accel_mss,speed_ms,0,blend_radius_m)
    speed_ms = 0.005
    movel([0.126015, -1.366636, -2.621765, -0.723988, 1.570796, 1.696812],accel_mss,speed_ms,0,blend_radius_m)
    speed_ms = 0.040
    # Splitting Linear movement in 6 (instruction 276: MoveL 187)
    movel([0.129480, -1.356816, -2.628292, -0.727281, 1.570796, 1.700277],accel_mss,speed_ms,0,blend_radius_m)
    movel([0.133025, -1.346823, -2.634791, -0.730775, 1.570796, 1.703821],accel_mss,speed_ms,0,blend_radius_m)
    movel([0.136651, -1.336650, -2.641261, -0.734478, 1.570796, 1.707448],accel_mss,speed_ms,0,blend_radius_m)
    movel([0.140363, -1.326290, -2.647701, -0.738398, 1.570796, 1.711159],accel_mss,speed_ms,0,blend_radius_m)
    movel([0.144163, -1.315735, -2.654109, -0.742545, 1.570796, 1.714959],accel_mss,speed_ms,0,blend_radius_m)
    movel([0.148054, -1.304976, -2.660485, -0.746928, 1.570796, 1.718851],accel_mss,speed_ms,0,blend_radius_m)
    speed_ms = 0.005
    movel([0.148054, -1.315442, -2.664697, -0.732250, 1.570796, 1.718851],accel_mss,speed_ms,0,blend_radius_m)
    speed_ms = 0.035
    # Splitting Linear movement in 2 (instruction 280: MoveL 189)
    movel([0.140988, -1.315968, -2.664384, -0.732038, 1.570796, 1.711785],accel_mss,speed_ms,0,blend_radius_m)
    movel([0.133907, -1.316541, -2.664042, -0.731806, 1.570796, 1.704703],accel_mss,speed_ms,0,blend_radius_m)
    movel([0.121536, -1.322360, -2.660548, -0.729481, 1.570796, 1.692332],accel_mss,speed_ms,0,blend_radius_m)
    movel([0.110994, -1.331121, -2.655199, -0.726068, 1.570796, 1.681791],accel_mss,speed_ms,0,blend_radius_m)
    movel([0.103432, -1.341492, -2.648729, -0.722168, 1.570796, 1.674229],accel_mss,speed_ms,0,blend_radius_m)
    movel([0.099878, -1.352233, -2.641865, -0.718291, 1.570796, 1.670674],accel_mss,speed_ms,0,blend_radius_m)
    movel([0.101046, -1.361360, -2.635902, -0.715127, 1.570796, 1.671842],accel_mss,speed_ms,0,blend_radius_m)
    movel([0.106376, -1.367425, -2.631872, -0.713092, 1.570796, 1.677172],accel_mss,speed_ms,0,blend_radius_m)
    movel([0.114967, -1.370059, -2.630105, -0.712225, 1.570796, 1.685764],accel_mss,speed_ms,0,blend_radius_m)
    movel([0.126042, -1.368817, -2.630939, -0.712633, 1.570796, 1.696838],accel_mss,speed_ms,0,blend_radius_m)
    speed_ms = 0.005
    movel([0.126042, -1.358805, -2.626981, -0.726602, 1.570796, 1.696838],accel_mss,speed_ms,0,blend_radius_m)
    speed_ms = 0.040
    # Splitting Linear movement in 8 (instruction 292: MoveL 199)
    movel([0.130470, -1.349010, -2.633381, -0.729998, 1.570796, 1.701267],accel_mss,speed_ms,0,blend_radius_m)
    movel([0.134997, -1.339040, -2.639754, -0.733595, 1.570796, 1.705793],accel_mss,speed_ms,0,blend_radius_m)
    movel([0.139626, -1.328890, -2.646099, -0.737400, 1.570796, 1.710422],accel_mss,speed_ms,0,blend_radius_m)
    movel([0.144360, -1.318551, -2.652414, -0.741424, 1.570796, 1.715157],accel_mss,speed_ms,0,blend_radius_m)
    movel([0.149204, -1.308016, -2.658699, -0.745674, 1.570796, 1.720001],accel_mss,speed_ms,0,blend_radius_m)
    movel([0.154162, -1.297276, -2.664953, -0.750160, 1.570796, 1.724958],accel_mss,speed_ms,0,blend_radius_m)
    movel([0.159237, -1.286322, -2.671175, -0.754892, 1.570796, 1.730033],accel_mss,speed_ms,0,blend_radius_m)
    movel([0.164434, -1.275146, -2.677362, -0.759881, 1.570796, 1.735230],accel_mss,speed_ms,0,blend_radius_m)
    speed_ms = 0.005
    movel([0.164434, -1.285840, -2.681716, -0.744833, 1.570796, 1.735230],accel_mss,speed_ms,0,blend_radius_m)
    speed_ms = 0.035
    movel([0.170344, -1.289502, -2.679674, -0.743213, 1.570796, 1.741140],accel_mss,speed_ms,0,blend_radius_m)
    movel([0.170362, -1.296066, -2.675969, -0.740354, 1.570796, 1.741159],accel_mss,speed_ms,0,blend_radius_m)
    movel([0.162120, -1.308070, -2.669045, -0.735274, 1.570796, 1.732916],accel_mss,speed_ms,0,blend_radius_m)
    speed_ms = 0.005
    movel([0.162120, -1.297546, -2.664798, -0.750045, 1.570796, 1.732916],accel_mss,speed_ms,0,blend_radius_m)
    speed_ms = 0.040
    # Splitting Linear movement in 4 (instruction 302: MoveL 205)
    movel([0.157415, -1.291782, -2.668093, -0.752514, 1.570796, 1.728212],accel_mss,speed_ms,0,blend_radius_m)
    movel([0.152634, -1.286018, -2.671345, -0.755026, 1.570796, 1.723430],accel_mss,speed_ms,0,blend_radius_m)
    movel([0.147774, -1.280255, -2.674554, -0.757581, 1.570796, 1.718571],accel_mss,speed_ms,0,blend_radius_m)
    movel([0.142835, -1.274494, -2.677718, -0.760177, 1.570796, 1.713631],accel_mss,speed_ms,0,blend_radius_m)
    speed_ms = 0.005
    movel([0.142835, -1.285192, -2.682076, -0.745121, 1.570796, 1.713631],accel_mss,speed_ms,0,blend_radius_m)
    speed_ms = 0.035
    movel([0.146098, -1.288335, -2.680327, -0.743727, 1.570796, 1.716894],accel_mss,speed_ms,0,blend_radius_m)
    movel([0.150281, -1.286148, -2.681545, -0.744696, 1.570796, 1.721078],accel_mss,speed_ms,0,blend_radius_m)
    movel([0.152811, -1.281988, -2.683846, -0.746555, 1.570796, 1.723607],accel_mss,speed_ms,0,blend_radius_m)
    speed_ms = 0.005
    movel([0.152811, -1.271267, -2.679472, -0.761650, 1.570796, 1.723607],accel_mss,speed_ms,0,blend_radius_m)
    speed_ms = 0.040
    # Splitting Linear movement in 4 (instruction 312: MoveL 211)
    movel([0.143399, -1.278371, -2.675593, -0.758425, 1.570796, 1.714195],accel_mss,speed_ms,0,blend_radius_m)
    movel([0.134099, -1.285422, -2.671679, -0.755288, 1.570796, 1.704895],accel_mss,speed_ms,0,blend_radius_m)
    movel([0.124910, -1.292418, -2.667731, -0.752239, 1.570796, 1.695706],accel_mss,speed_ms,0,blend_radius_m)
    movel([0.115831, -1.299362, -2.663750, -0.749277, 1.570796, 1.686628],accel_mss,speed_ms,0,blend_radius_m)
    speed_ms = 0.005
    movel([0.115831, -1.309872, -2.667989, -0.734528, 1.570796, 1.686628],accel_mss,speed_ms,0,blend_radius_m)
    speed_ms = 0.035
    movel([0.119018, -1.311663, -2.666935, -0.733791, 1.570796, 1.689815],accel_mss,speed_ms,0,blend_radius_m)
    movel([0.124552, -1.308327, -2.668895, -0.735167, 1.570796, 1.695349],accel_mss,speed_ms,0,blend_radius_m)
    movel([0.128682, -1.302365, -2.672360, -0.737664, 1.570796, 1.699479],accel_mss,speed_ms,0,blend_radius_m)
    movel([0.137107, -1.296040, -2.675984, -0.740365, 1.570796, 1.707904],accel_mss,speed_ms,0,blend_radius_m)
    movel([0.147439, -1.294947, -2.676605, -0.740837, 1.570796, 1.718235],accel_mss,speed_ms,0,blend_radius_m)
    movel([0.154749, -1.291993, -2.678275, -0.742121, 1.570796, 1.725546],accel_mss,speed_ms,0,blend_radius_m)
    movel([0.158291, -1.287522, -2.680780, -0.744086, 1.570796, 1.729087],accel_mss,speed_ms,0,blend_radius_m)
    movel([0.159480, -1.281108, -2.684330, -0.746952, 1.570796, 1.730276],accel_mss,speed_ms,0,blend_radius_m)
    speed_ms = 0.005
    # Splitting Linear movement in 4 (instruction 325: MoveL 221)
    movel([0.159480, -1.267736, -2.678848, -0.765805, 1.570796, 1.730276],accel_mss,speed_ms,0,blend_radius_m)
    movel([0.159480, -1.254747, -2.673268, -0.784374, 1.570796, 1.730276],accel_mss,speed_ms,0,blend_radius_m)
    movel([0.159480, -1.242136, -2.667592, -0.802661, 1.570796, 1.730276],accel_mss,speed_ms,0,blend_radius_m)
    movel([0.159480, -1.229897, -2.661823, -0.820668, 1.570796, 1.730276],accel_mss,speed_ms,0,blend_radius_m)
    speed_ms = 1.000
    movel([0.159480, -1.229897, -2.661823, -0.820668, 1.570796, 1.730276],accel_mss,speed_ms,0,blend_radius_m)
    # Splitting Linear movement in 22 (instruction 328: MoveL 223)
    movel([0.159480, -1.219089, -2.656501, -0.836799, 1.570796, 1.730276],accel_mss,speed_ms,0,blend_radius_m)
    movel([0.159480, -1.208578, -2.651107, -0.852704, 1.570796, 1.730276],accel_mss,speed_ms,0,blend_radius_m)
    movel([0.159480, -1.198359, -2.645642, -0.868387, 1.570796, 1.730276],accel_mss,speed_ms,0,blend_radius_m)
    movel([0.159480, -1.188429, -2.640110, -0.883850, 1.570796, 1.730276],accel_mss,speed_ms,0,blend_radius_m)
    movel([0.159480, -1.178781, -2.634511, -0.899097, 1.570796, 1.730276],accel_mss,speed_ms,0,blend_radius_m)
    movel([0.159480, -1.169410, -2.628848, -0.914131, 1.570796, 1.730276],accel_mss,speed_ms,0,blend_radius_m)
    movel([0.159480, -1.160312, -2.623122, -0.928955, 1.570796, 1.730276],accel_mss,speed_ms,0,blend_radius_m)
    movel([0.159480, -1.151481, -2.617334, -0.943574, 1.570796, 1.730276],accel_mss,speed_ms,0,blend_radius_m)
    movel([0.159480, -1.142911, -2.611488, -0.957990, 1.570796, 1.730276],accel_mss,speed_ms,0,blend_radius_m)
    movel([0.159480, -1.134598, -2.605584, -0.972207, 1.570796, 1.730276],accel_mss,speed_ms,0,blend_radius_m)
    movel([0.159480, -1.126536, -2.599623, -0.986230, 1.570796, 1.730276],accel_mss,speed_ms,0,blend_radius_m)
    movel([0.159480, -1.118720, -2.593607, -1.000061, 1.570796, 1.730276],accel_mss,speed_ms,0,blend_radius_m)
    movel([0.159480, -1.111145, -2.587538, -1.013706, 1.570796, 1.730276],accel_mss,speed_ms,0,blend_radius_m)
    movel([0.159480, -1.103806, -2.581417, -1.027166, 1.570796, 1.730276],accel_mss,speed_ms,0,blend_radius_m)
    movel([0.159480, -1.096697, -2.575245, -1.040447, 1.570796, 1.730276],accel_mss,speed_ms,0,blend_radius_m)
    movel([0.159480, -1.089814, -2.569023, -1.053552, 1.570796, 1.730276],accel_mss,speed_ms,0,blend_radius_m)
    movel([0.159480, -1.083151, -2.562753, -1.066485, 1.570796, 1.730276],accel_mss,speed_ms,0,blend_radius_m)
    movel([0.159480, -1.076704, -2.556435, -1.079249, 1.570796, 1.730276],accel_mss,speed_ms,0,blend_radius_m)
    movel([0.159480, -1.070468, -2.550072, -1.091849, 1.570796, 1.730276],accel_mss,speed_ms,0,blend_radius_m)
    movel([0.159480, -1.064439, -2.543663, -1.104287, 1.570796, 1.730276],accel_mss,speed_ms,0,blend_radius_m)
    movel([0.159480, -1.058610, -2.537210, -1.116569, 1.570796, 1.730276],accel_mss,speed_ms,0,blend_radius_m)
    movel([0.159480, -1.052979, -2.530714, -1.128696, 1.570796, 1.730276],accel_mss,speed_ms,0,blend_radius_m)
    # End of main program
  end

  Machining1()
end
